{attribute 'GeneratedUsingTerminal: EL2521-0124-0016'}
{attribute addProperty BoxType "EL2521-0124-0016"}
{attribute addProperty Id "Enable_latch_extern_on_positive_edgeAT %Q*BOOL1Set_counterAT %Q*BOOL1Enable_latch_extern_on_negative_edgeAT %Q*BOOL1Set_counter_valueAT %Q*UINT2"}
{attribute addProperty CRC "3696109835"}
{attribute addProperty Size "5"}
TYPE ENC_Control_compact_DC4E290B :
STRUCT
	{attribute addProperty Name "Enable_latch_extern_on_positive_edge"}
	Enable_latch_extern_on_positive_edge AT %Q* : BOOL;
	{attribute addProperty Name "Set_counter"}
	Set_counter AT %Q* : BOOL;
	{attribute addProperty Name "Enable_latch_extern_on_negative_edge"}
	Enable_latch_extern_on_negative_edge AT %Q* : BOOL;
	{attribute addProperty Name "Set_counter_value"}
	Set_counter_value AT %Q* : UINT;
END_STRUCT
END_TYPE

(* stored: Version 1.2.0.0, ProductVersion 3.1.4024.9
   DUT ENC_Control_compact_DC4E290B: Id {52f293b2-1264-4ff9-8b2a-e30da871d8a0} *)
